{attribute addProperty BoxType "EK1100-0000-0018"}
{attribute addProperty Id "Beckhoff_AX2xxxEK1122Beckhoff_AX2xxxEK1122_F89967F723229"}
{attribute addProperty CRC "643680986"}
{attribute addProperty SizeInBites "232"}
{attribute addProperty SizeInBytes "29"}
TYPE Beckhoff_AX2xxx_265DCADA EXTENDS EK1100_179A0949 :
STRUCT
	{attribute addProperty Name "Beckhoff_AX2xxxEK1122"}
	Beckhoff_AX2xxxEK1122 : Beckhoff_AX2xxxEK1122_F89967F7;
END_STRUCT
END_TYPE

(* stored: Version 1.2.0.0, ProductVersion 3.1.4024.9
   DUT Beckhoff_AX2xxx_265DCADA: Id {620fe7da-4dfd-4c7a-9261-e6203fcbc834} *)
